FUNCTION_BLOCK serializeLrealArray2ByteArray (* Basic Function Block Type *)
  (* Standard: 61499-2 *)
  (* Version 0.0, 19/09/2015, kollger, nxtControl GmbH, Template *)
  PACKAGE Main;
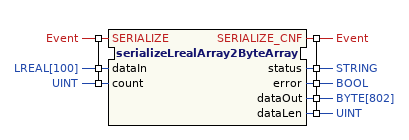
  EVENT_INPUT
    SERIALIZE WITH dataIn, count; (* Normal Execution Request *)
  END_EVENT
  EVENT_OUTPUT
    SERIALIZE_CNF WITH dataOut, dataLen, status, error; (* Execution Confirmation *)
  END_EVENT
  VAR_INPUT
    dataIn : ARRAY [0..99] OF LREAL;
    count : UINT;
  END_VAR
  VAR_OUTPUT
    status : STRING;
    error : BOOL;
    dataOut : ARRAY [0..801] OF BYTE;
    dataLen : UINT;
  END_VAR
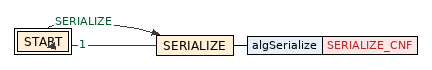
  EC_STATES
    START; (* Initial State *)
    SERIALIZE : algSerialize -> SERIALIZE_CNF; (* Normal execution *)
  END_STATES
  EC_TRANSITIONS
    START TO SERIALIZE := SERIALIZE;
    SERIALIZE TO START := 1;
  END_TRANSITIONS
  ALGORITHM algSerialize IN ST: (* Normally executed algorithm *)
VAR
	index : UINT := 0;
	byteindex : UINT := 0;
	varLWORD : LWORD := 16#0;
END_VAR;

IF count <= 100 THEN

	(* Iterate through the LREAL array and transfer it to the BYTE ARRAY *)
	FOR index := 0 TO count - 1 DO
		varLWORD := LREAL_TO_LWORD(dataIn[index]);
		byteindex := index * 8 + 2;
		dataOut[byteindex] := LWORD_TO_BYTE(ROR(varLWORD,56));
		dataOut[byteindex + 1] := LWORD_TO_BYTE(ROR(varLWORD,48));
		dataOut[byteindex + 2] := LWORD_TO_BYTE(ROR(varLWORD,40));
		dataOut[byteindex + 3] := LWORD_TO_BYTE(ROR(varLWORD,32));
		dataOut[byteindex + 4] := LWORD_TO_BYTE(ROR(varLWORD,24));
		dataOut[byteindex + 5] := LWORD_TO_BYTE(ROR(varLWORD,16));
		dataOut[byteindex + 6] := LWORD_TO_BYTE(ROR(varLWORD,8));
		dataOut[byteindex + 7] := LWORD_TO_BYTE(varLWORD);
	END_FOR;

	(* calculate data length *)
	dataLen := count * 8 + 2;

	(* encode data length *)
	dataOut[0] := WORD_TO_BYTE(ROR(UINT_TO_WORD(count),8));
	dataOut[1] := WORD_TO_BYTE(UINT_TO_WORD(count));

  error := FALSE;
  status := STRING#'Ok';
ELSE
  error := TRUE;
  status := STRING#'count to big';
END_IF;
  END_ALGORITHM
END_FUNCTION_BLOCK
